PROGRAM OP10A_Camera_FB
VAR
	OP10A_LH_Camera 			        : FB_Cognex_ProfiNET_1;
	
	OP10A_LH_Acquisition_Status AT %I*    :Acquisition_Status;
	OP10A_LH_Inspection_Status  AT %I*    :Inspection_Status;	
	OP10A_LH_Acquisition_ID     AT %I*    :UINT;
	OP10A_LH_Inspection_ID   	 AT %I*  :UINT;
	OP10A_LH_Error_code      	 AT %I*  :UINT;
	OP10A_LH_Current_Job_ID  	 AT %I*  :UINT;
	OP10A_LH_Result_code     	 AT %I*  :UINT;
	OP10A_LH_Cam_Result      	 AT %I*  :ARRAY[0..63] OF BYTE;	
	OP10A_LH_Acquisition_Control AT %Q*  : Acquisition_Control;
	OP10A_LH_Inspection_Control  AT %Q*  : Inspection_Control;
	OP10A_LH_Command_word		AT %Q*  : UINT;
	OP10A_LH_Union                       : UNION_64Byte;

	OP10A_RH_Camera 			          : FB_Cognex_ProfiNET_1;

	
	OP10A_RH_Acquisition_Status AT %I*    :Acquisition_Status;
	OP10A_RH_Inspection_Status  AT %I*    :Inspection_Status;	
	OP10A_RH_Acquisition_ID     AT %I*    :UINT;
	OP10A_RH_Inspection_ID   	 AT %I*  :UINT;
	OP10A_RH_Error_code      	 AT %I*  :UINT;
	OP10A_RH_Current_Job_ID  	 AT %I*  :UINT;
	OP10A_RH_Result_code     	 AT %I*  :UINT;
	OP10A_RH_Cam_Result      	 AT %I*  :ARRAY[0..63] OF BYTE;	
	OP10A_RH_Acquisition_Control AT %Q*  : Acquisition_Control;
	OP10A_RH_Inspection_Control  AT %Q*  : Inspection_Control;
	OP10A_RH_Command_word		AT %Q*  : UINT;
	OP10A_RH_Union                       : UNION_64Byte;
	
	OP10_A_Empty_Camera_1	      : FB_Cognex_ProfiNET_1;
	
	
	OP10A_Empty_Cam_1_Acquisition_Status   AT %I*  :Acquisition_Status;
	OP10A_Empty_Cam_1_Inspection_Status    AT %I*  :Inspection_Status;	
	OP10A_Empty_Cam_1_Acquisition_ID       AT %I*  :UINT;
	OP10A_Empty_Cam_1_Inspection_ID   	 AT %I*  :UINT;
	OP10A_Empty_Cam_1_Error_code      	 AT %I*  :UINT;
	OP10A_Empty_Cam_1_Current_Job_ID  	 AT %I*  :UINT;
	OP10A_Empty_Cam_1_Result_code     	 AT %I*  :UINT;
	OP10A_Empty_Cam_1_Result      	 AT %I*  :ARRAY[0..63] OF BYTE;
	
	OP10A_Empty_Cam_1_Acquisition_Control AT %Q*  : Acquisition_Control;
	OP10A_Empty_Cam_1_Inspection_Control  AT %Q*  : Inspection_Control;
	OP10A_Empty_Cam_1_Command_word		AT %Q*  : UINT;
	Error_status_Cam_1						      : STRING;
	OP10A_Empty_Cam_1_Target_Job_ID				  : UINT;
	OP10A_Empty_Cam_1_Loaded_Job_ID		    	  : UINT;
	OP10A_Empty_Cam_1_Union                       : UNION_64Byte;
	OP10A_Empty_Cam_1_Job_Change_Complete		  : BOOL;
	OP10A_Empty_Cam_1_Job_Change_Error   		  : BOOL;
	OP10A_Empty_Cam_1_Picture_Taken      		  : BOOL;	
	
END_VAR

OP10A_LH_Camera (
	tTimeout:= , 
	sJob_Name:= , 
	camera_ready=> OP10A_LH_Camera_Ready,
	Camera_online=> OP10A_LH_Camera_Online,
	stCognex_record_status:=OP10A_LH_Acquisition_Status, 
	Acquisition_ID:=OP10A_LH_Acquisition_ID , 
	stCognex_Inspection_status:=OP10A_LH_Inspection_Status, 
	Error_Code:=OP10A_LH_Error_code , 
	wcommand_control_in:= OP10A_LH_Current_Job_ID, 
	aResults_64_Bytes:= OP10A_LH_Cam_Result, 
	number_of_inspections:=OP10A_LH_Inspection_ID , 
	iresult_code:= OP10A_LH_Result_code, 
	bTarget_job_ID:=OP10A_LH_Target_Job_ID , 
	Error_Status_message=> OP10A_LH_Error_status, 
	bError=> OP10A_LH_Camera_Error, 
	stCognex_record_control=>OP10A_LH_Acquisition_Control , 
	stCognex_inspection_control=>OP10A_LH_Inspection_Control , 
	wCommandControl_out=>OP10A_LH_Command_word , 
	aUser_data_64_Byte=> OP10A_LH_Union.aArrayOfByte, 
	bJob_loading_completed=>OP10A_LH_Job_Change_Complete , 
	bJob_load_failed=>OP10A_LH_Job_Change_Error , 
	bInspection_Result_IO=>  , 
	bInspection_Result_NIO=> , 
	bTXTSM_Error_Job_Change=> OP10A_LH_Job_Change_Error, 
	bPictureTakenComplete=> OP10A_LH_Picture_Taken, 
	Loaded_Job_ID=>OP10A_LH_Loaded_Job_ID	 , 
	bClear_Error:= HMI_Reset, 
	bJob_change_start:= OP10A_LH_Camera_Job_Change_start, 
	TXTSM_camera_not_online=>OP10A_LH_Camera_Error	 , 
	bTrigger_start:= OP10A_LH_Camera_Trigger );
	
OP10A_RH_Camera (
	tTimeout:= , 
	sJob_Name:= , 
	camera_ready=> OP10A_RH_Camera_Ready,
	Camera_online=> OP10A_RH_Camera_Online,
	stCognex_record_status:=OP10A_RH_Acquisition_Status, 
	Acquisition_ID:=OP10A_RH_Acquisition_ID , 
	stCognex_Inspection_status:=OP10A_RH_Inspection_Status, 
	Error_Code:=OP10A_RH_Error_code , 
	wcommand_control_in:= OP10A_RH_Current_Job_ID, 
	aResults_64_Bytes:= OP10A_RH_Cam_Result, 
	number_of_inspections:=OP10A_RH_Inspection_ID , 
	iresult_code:= OP10A_RH_Result_code, 
	bTarget_job_ID:=OP10A_RH_Target_Job_ID , 
	Error_Status_message=> OP10A_RH_Error_status, 
	bError=> OP10A_RH_Camera_Error, 
	stCognex_record_control=>OP10A_RH_Acquisition_Control , 
	stCognex_inspection_control=>OP10A_RH_Inspection_Control , 
	wCommandControl_out=>OP10A_RH_Command_word , 
	aUser_data_64_Byte=> OP10A_RH_Union.aArrayOfByte, 
	bJob_loading_completed=>OP10A_RH_Job_Change_Complete , 
	bJob_load_failed=>OP10A_RH_Job_Change_Error , 
	bInspection_Result_IO=>  , 
	bInspection_Result_NIO=> , 
	bTXTSM_Error_Job_Change=> OP10A_RH_Job_Change_Error, 
	bPictureTakenComplete=> OP10A_RH_Picture_Taken, 
	Loaded_Job_ID=>OP10A_RH_Loaded_Job_ID	 , 
	bClear_Error:= HMI_Reset, 
	bJob_change_start:= OP10A_RH_Camera_Job_Change_start, 
	TXTSM_camera_not_online=>OP10A_RH_Camera_Error	 , 
	bTrigger_start:= OP10A_RH_Camera_Trigger );	
	
OP10_A_Empty_Camera_1(
	tTimeout:= , 
	sJob_Name:= , 
	camera_ready=> OP10A_Empty_Cam_1_Camera_Ready,
	Camera_online=> OP10A_Empty_Cam_1_Camera_Online,
	stCognex_record_status:=OP10A_Empty_Cam_1_Acquisition_Status, 
	Acquisition_ID:=OP10A_Empty_Cam_1_Acquisition_ID , 
	stCognex_Inspection_status:=OP10A_Empty_Cam_1_Inspection_Status, 
	Error_Code:=OP10A_Empty_Cam_1_Error_code , 
	wcommand_control_in:= OP10A_Empty_Cam_1_Current_Job_ID, 
	aResults_64_Bytes:= OP10A_Empty_Cam_1_Result, 
	number_of_inspections:=OP10A_Empty_Cam_1_Inspection_ID , 
	iresult_code:= OP10A_Empty_Cam_1_Result_code, 
	bTarget_job_ID:=OP10A_Empty_Cam_1_Target_Job_ID , 
	Error_Status_message=> Error_status_Cam_1, 
	bError=> OP10A_Empty_Cam_1_Camera_Error, 
	stCognex_record_control=>OP10A_Empty_Cam_1_Acquisition_Control , 
	stCognex_inspection_control=>OP10A_Empty_Cam_1_Inspection_Control , 
	wCommandControl_out=>OP10A_Empty_Cam_1_Command_word , 
	aUser_data_64_Byte=> OP10A_Empty_Cam_1_Union.aArrayOfByte, 
	bJob_loading_completed=>OP10A_Empty_Cam_1_Job_Change_Complete, 
	bJob_load_failed=>OP10A_Empty_Cam_1_Job_Change_Error , 
	bInspection_Result_IO=>  , 
	bInspection_Result_NIO=> , 
	bTXTSM_Error_Job_Change=> OP10A_Empty_Cam_1_Job_Change_Error, 
	bPictureTakenComplete=> OP10A_Empty_Cam_1_Picture_Taken, 
	Loaded_Job_ID=>OP10A_Empty_Cam_1_Loaded_Job_ID	 , 
	bClear_Error:= HMI_Reset, 
	bJob_change_start:= OP10A_Empty_Cam_1_Camera_Job_Change_start, 
	TXTSM_camera_not_online=>OP10A_Empty_Cam_1_Camera_Error	 , 
	bTrigger_start:= OP10A_Empty_Cam_1_Camera_Trigger );

END_PROGRAM

(* stored: Version 1.1.0.1, ProductVersion 3.1.4024.11
   POU OP10A_Camera_FB: Id {585b0f78-3dda-41bb-b22a-da4b509b0a14}, SpecialFunc None *)
